Fanuc TP program (LS listing): block_2R_B2_4_Q40_R10.ls

/PROG  block_2R_B2_4_Q40_R10
/ATTR
COMMENT	= "19-04-12 14:24:10";
PROG_SIZE	= 0;
DEFAULT_GROUP	= 1, *, *, *, *;
/APPL
    ARC Welding Equipment: 1, *, *, *, *;
/MN
   1:  CALL HOME_ALL;
   1:  UFRAME_NUM = 1;
   1:  UTOOL_NUM = 3;
   1:  COL GUARD ADJUST 150;
   1:  !Teach Startpoint in PR90;
   1:  !Weld speed R100 in mm/sec;
   1:  !Retraction +Z in R101 in mm;
   1:  !Retraction speed in R102 in %;
   1:  !END_PUB Time in R103;
   1:  !Zeit bis Drahtvorschub R104;
   1:  !Drahtvorschubzeit R105;
   1:  !- Layer/Ebene 1;
   1:  PR[91] = PR[90];
   1:  PR[91,1] = PR[90,1] + 38.877;
   1:  PR[91,2] = PR[90,2] + 1.192;
   1:  PR[91,3] = PR[90,3] + 2.500;
   1:  PR[92] = PR[91];
   1:  PR[92,3] = PR[92,3] + R[101];
   1:J PR[92] R[102]% CNT100;
   1:L PR[91] 100mm/sec FINE RampTo R[100]  Weld Start[1,5.0];
   1:  GO[2]=R[111];
   1:  PR[91,2] = PR[90,2] + 38.792;
   1:L PR[91] R[100]mm/sec CNT100;
   1:  PR[91,1] = PR[90,1] + 1.277;
   1:L PR[91] R[100]mm/sec CNT100;
   1:  PR[91,2] = PR[90,2] + 1.192;
   1:L PR[91] R[100]mm/sec CNT100;
   1:  PR[91,1] = PR[90,1] + 38.877;
   1:L PR[91] R[100]mm/sec CNT100  Weld End[1,5.0,0.2s];
   1:  WAIT R[104];
   1:  PR[92] = PR[91];
   1:  PR[92,3] = PR[92,3] + R[101];
   1:J PR[92] R[102]% CNT100;
   1:  PR[91,1] = PR[90,1] + 36.477;
   1:  PR[91,2] = PR[90,2] + 3.592;
   1:  PR[92] = PR[91];
   1:  PR[92,3] = PR[92,3] + R[101];
   1:J PR[92] R[102]% CNT100;
   1:L PR[91] 100mm/sec FINE RampTo R[100]  Weld Start[1,5.0];
   1:  GO[2]=R[111];
   1:  PR[91,2] = PR[90,2] + 36.392;
   1:L PR[91] R[100]mm/sec CNT100;
   1:  PR[91,1] = PR[90,1] + 3.677;
   1:L PR[91] R[100]mm/sec CNT100;
   1:  PR[91,2] = PR[90,2] + 3.592;
   1:L PR[91] R[100]mm/sec CNT100;
   1:  PR[91,1] = PR[90,1] + 36.477;
   1:L PR[91] R[100]mm/sec CNT100  Weld End[1,5.0,0.2s];
   1:  WAIT R[104];
   1:  PR[92] = PR[91];
   1:  PR[92,3] = PR[92,3] + R[101];
   1:J PR[92] R[102]% CNT100;
   1:  PR[91,1] = PR[90,1] + 25.483;
   1:  PR[91,2] = PR[90,2] + 16.870;
   1:  PR[92] = PR[91];
   1:  PR[92,3] = PR[92,3] + R[101];
   1:J PR[92] R[102]% CNT100;
   1:L PR[91] 100mm/sec FINE RampTo R[100]  Weld Start[1,5.0];
   1:  GO[2]=R[111];
   1:  PR[91,1] = PR[90,1] + 23.198;
   1:  PR[91,2] = PR[90,2] + 14.586;
   1:L PR[91] R[100]mm/sec CNT100;
   1:  PR[91,1] = PR[90,1] + 20.077;
   1:  PR[91,2] = PR[90,2] + 13.750;
   1:L PR[91] R[100]mm/sec CNT100;
   1:  PR[91,1] = PR[90,1] + 16.957;
   1:  PR[91,2] = PR[90,2] + 14.586;
   1:L PR[91] R[100]mm/sec CNT100;
   1:  PR[91,1] = PR[90,1] + 14.672;
   1:  PR[91,2] = PR[90,2] + 16.870;
   1:L PR[91] R[100]mm/sec CNT100;
   1:  PR[91,1] = PR[90,1] + 13.835;
   1:  PR[91,2] = PR[90,2] + 19.992;
   1:L PR[91] R[100]mm/sec CNT100;
   1:  PR[91,1] = PR[90,1] + 14.672;
   1:  PR[91,2] = PR[90,2] + 23.113;
   1:L PR[91] R[100]mm/sec CNT100;
   1:  PR[91,1] = PR[90,1] + 16.957;
   1:  PR[91,2] = PR[90,2] + 25.398;
   1:L PR[91] R[100]mm/sec CNT100;
   1:  PR[91,1] = PR[90,1] + 20.077;
   1:  PR[91,2] = PR[90,2] + 26.234;
   1:L PR[91] R[100]mm/sec CNT100;
   1:  PR[91,1] = PR[90,1] + 23.198;
   1:  PR[91,2] = PR[90,2] + 25.398;
   1:L PR[91] R[100]mm/sec CNT100;
   1:  PR[91,1] = PR[90,1] + 25.483;
   1:  PR[91,2] = PR[90,2] + 23.113;
   1:L PR[91] R[100]mm/sec CNT100;
   1:  PR[91,1] = PR[90,1] + 26.320;
   1:  PR[91,2] = PR[90,2] + 19.992;
   1:L PR[91] R[100]mm/sec CNT100;
   1:  PR[91,1] = PR[90,1] + 25.483;
   1:  PR[91,2] = PR[90,2] + 16.870;
   1:L PR[91] R[100]mm/sec CNT100  Weld End[1,5.0,0.2s];
   1:  WAIT R[104];
   1:  PR[92] = PR[91];
   1:  PR[92,3] = PR[92,3] + R[101];
   1:J PR[92] R[102]% CNT100;
   1:  PR[91,1] = PR[90,1] + 27.635;
   1:  PR[91,2] = PR[90,2] + 15.627;
   1:  PR[92] = PR[91];
   1:  PR[92,3] = PR[92,3] + R[101];
   1:J PR[92] R[102]% CNT100;
   1:L PR[91] 100mm/sec FINE RampTo R[100]  Weld Start[1,5.0];
   1:  GO[2]=R[111];
   1:  PR[91,1] = PR[90,1] + 24.440;
   1:  PR[91,2] = PR[90,2] + 12.434;
   1:L PR[91] R[100]mm/sec CNT100;
   1:  PR[91,1] = PR[90,1] + 20.077;
   1:  PR[91,2] = PR[90,2] + 11.265;
   1:L PR[91] R[100]mm/sec CNT100;
   1:  PR[91,1] = PR[90,1] + 15.715;
   1:  PR[91,2] = PR[90,2] + 12.434;
   1:L PR[91] R[100]mm/sec CNT100;
   1:  PR[91,1] = PR[90,1] + 12.520;
   1:  PR[91,2] = PR[90,2] + 15.627;
   1:L PR[91] R[100]mm/sec CNT100;
   1:  PR[91,1] = PR[90,1] + 11.350;
   1:  PR[91,2] = PR[90,2] + 19.992;
   1:L PR[91] R[100]mm/sec CNT100;
   1:  PR[91,1] = PR[90,1] + 12.520;
   1:  PR[91,2] = PR[90,2] + 24.356;
   1:L PR[91] R[100]mm/sec CNT100;
   1:  PR[91,1] = PR[90,1] + 15.715;
   1:  PR[91,2] = PR[90,2] + 27.550;
   1:L PR[91] R[100]mm/sec CNT100;
   1:  PR[91,1] = PR[90,1] + 20.077;
   1:  PR[91,2] = PR[90,2] + 28.719;
   1:L PR[91] R[100]mm/sec CNT100;
   1:  PR[91,1] = PR[90,1] + 24.440;
   1:  PR[91,2] = PR[90,2] + 27.550;
   1:L PR[91] R[100]mm/sec CNT100;
   1:  PR[91,1] = PR[90,1] + 27.635;
   1:  PR[91,2] = PR[90,2] + 24.356;
   1:L PR[91] R[100]mm/sec CNT100;
   1:  PR[91,1] = PR[90,1] + 28.805;
   1:  PR[91,2] = PR[90,2] + 19.992;
   1:L PR[91] R[100]mm/sec CNT100;
   1:  PR[91,1] = PR[90,1] + 27.635;
   1:  PR[91,2] = PR[90,2] + 15.627;
   1:L PR[91] R[100]mm/sec CNT100  Weld End[1,5.0,0.2s];
   1:  WAIT R[104];
   1:  PR[92] = PR[91];
   1:  PR[92,3] = PR[92,3] + R[101];
   1:J PR[92] R[102]% CNT100;
   1:  PR[91,1] = PR[90,1] + 29.744;
   1:  PR[91,2] = PR[90,2] + 16.082;
   1:  PR[92] = PR[91];
   1:  PR[92,3] = PR[92,3] + R[101];
   1:J PR[92] R[102]% CNT100;
   1:L PR[91] 100mm/sec FINE RampTo R[100]  Weld Start[1,5.0];
   1:  GO[2]=R[111];
   1:  PR[91,1] = PR[90,1] + 34.557;
   1:  PR[91,2] = PR[90,2] + 20.895;
   1:L PR[91] R[100]mm/sec CNT100;
   1:  PR[91,2] = PR[90,2] + 24.289;
   1:L PR[91] R[100]mm/sec CNT100;
   1:  PR[91,1] = PR[90,1] + 30.680;
   1:  PR[91,2] = PR[90,2] + 20.412;
   1:L PR[91] R[100]mm/sec CNT100;
   1:  PR[91,1] = PR[90,1] + 29.962;
   1:  PR[91,2] = PR[90,2] + 23.088;
   1:L PR[91] R[100]mm/sec CNT100;
   1:  PR[91,1] = PR[90,1] + 34.557;
   1:  PR[91,2] = PR[90,2] + 27.683;
   1:L PR[91] R[100]mm/sec CNT100;
   1:  PR[91,2] = PR[90,2] + 31.078;
   1:L PR[91] R[100]mm/sec CNT100;
   1:  PR[91,1] = PR[90,1] + 29.093;
   1:  PR[91,2] = PR[90,2] + 25.613;
   1:L PR[91] R[100]mm/sec CNT100;
   1:  PR[91,1] = PR[90,1] + 27.396;
   1:  PR[91,2] = PR[90,2] + 27.310;
   1:L PR[91] R[100]mm/sec CNT100;
   1:  PR[91,1] = PR[90,1] + 34.557;
   1:  PR[91,2] = PR[90,2] + 34.472;
   1:L PR[91] R[100]mm/sec CNT100;
   1:  PR[91,1] = PR[90,1] + 31.163;
   1:L PR[91] R[100]mm/sec CNT100;
   1:  PR[91,1] = PR[90,1] + 25.698;
   1:  PR[91,2] = PR[90,2] + 29.007;
   1:L PR[91] R[100]mm/sec CNT100;
   1:  PR[91,1] = PR[90,1] + 25.434;
   1:  PR[91,2] = PR[90,2] + 29.271;
   1:L PR[91] R[100]mm/sec CNT100;
   1:  PR[91,1] = PR[90,1] + 23.174;
   1:  PR[91,2] = PR[90,2] + 29.877;
   1:L PR[91] R[100]mm/sec CNT100;
   1:  PR[91,1] = PR[90,1] + 27.769;
   1:  PR[91,2] = PR[90,2] + 34.472;
   1:L PR[91] R[100]mm/sec CNT100;
   1:  PR[91,1] = PR[90,1] + 24.375;
   1:L PR[91] R[100]mm/sec CNT100;
   1:  PR[91,1] = PR[90,1] + 20.497;
   1:  PR[91,2] = PR[90,2] + 30.594;
   1:L PR[91] R[100]mm/sec CNT100  Weld End[1,5.0,0.2s];
   1:  WAIT R[104];
   1:  PR[92] = PR[91];
   1:  PR[92,3] = PR[92,3] + R[101];
   1:J PR[92] R[102]% CNT100;
   1:  PR[91,1] = PR[90,1] + 7.405;
   1:  PR[91,2] = PR[90,2] + 34.472;
   1:  PR[92] = PR[91];
   1:  PR[92,3] = PR[92,3] + R[101];
   1:J PR[92] R[102]% CNT100;
   1:L PR[91] 100mm/sec FINE RampTo R[100]  Weld Start[1,5.0];
   1:  GO[2]=R[111];
   1:  PR[91,1] = PR[90,1] + 5.597;
   1:  PR[91,2] = PR[90,2] + 32.665;
   1:L PR[91] R[100]mm/sec CNT100;
   1:  PR[91,2] = PR[90,2] + 29.270;
   1:L PR[91] R[100]mm/sec CNT100;
   1:  PR[91,1] = PR[90,1] + 10.799;
   1:  PR[91,2] = PR[90,2] + 34.472;
   1:L PR[91] R[100]mm/sec CNT100;
   1:  PR[91,1] = PR[90,1] + 14.193;
   1:L PR[91] R[100]mm/sec CNT100;
   1:  PR[91,1] = PR[90,1] + 5.597;
   1:  PR[91,2] = PR[90,2] + 25.876;
   1:L PR[91] R[100]mm/sec CNT100;
   1:  PR[91,2] = PR[90,2] + 22.482;
   1:L PR[91] R[100]mm/sec CNT100;
   1:  PR[91,1] = PR[90,1] + 17.587;
   1:  PR[91,2] = PR[90,2] + 34.472;
   1:L PR[91] R[100]mm/sec CNT100;
   1:  PR[91,1] = PR[90,1] + 20.981;
   1:L PR[91] R[100]mm/sec CNT100;
   1:  PR[91,1] = PR[90,1] + 16.168;
   1:  PR[91,2] = PR[90,2] + 29.659;
   1:L PR[91] R[100]mm/sec CNT100;
   1:  PR[91,1] = PR[90,1] + 14.721;
   1:  PR[91,2] = PR[90,2] + 29.271;
   1:L PR[91] R[100]mm/sec CNT100;
   1:  PR[91,1] = PR[90,1] + 10.799;
   1:  PR[91,2] = PR[90,2] + 25.350;
   1:L PR[91] R[100]mm/sec CNT100;
   1:  PR[91,1] = PR[90,1] + 10.410;
   1:  PR[91,2] = PR[90,2] + 23.901;
   1:L PR[91] R[100]mm/sec CNT100;
   1:  PR[91,1] = PR[90,1] + 5.597;
   1:  PR[91,2] = PR[90,2] + 19.088;
   1:L PR[91] R[100]mm/sec CNT100;
   1:  PR[91,2] = PR[90,2] + 15.694;
   1:L PR[91] R[100]mm/sec CNT100;
   1:  PR[91,1] = PR[90,1] + 9.475;
   1:  PR[91,2] = PR[90,2] + 19.572;
   1:L PR[91] R[100]mm/sec CNT100;
   1:  PR[91,1] = PR[90,1] + 10.193;
   1:  PR[91,2] = PR[90,2] + 16.895;
   1:L PR[91] R[100]mm/sec CNT100;
   1:  PR[91,1] = PR[90,1] + 5.597;
   1:  PR[91,2] = PR[90,2] + 12.300;
   1:L PR[91] R[100]mm/sec CNT100;
   1:  PR[91,2] = PR[90,2] + 8.906;
   1:L PR[91] R[100]mm/sec CNT100;
   1:  PR[91,1] = PR[90,1] + 11.062;
   1:  PR[91,2] = PR[90,2] + 14.370;
   1:L PR[91] R[100]mm/sec CNT100;
   1:  PR[91,1] = PR[90,1] + 12.759;
   1:  PR[91,2] = PR[90,2] + 12.673;
   1:L PR[91] R[100]mm/sec CNT100;
   1:  PR[91,1] = PR[90,1] + 5.597;
   1:  PR[91,2] = PR[90,2] + 5.512;
   1:L PR[91] R[100]mm/sec CNT100;
   1:  PR[91,1] = PR[90,1] + 8.992;
   1:L PR[91] R[100]mm/sec CNT100;
   1:  PR[91,1] = PR[90,1] + 14.456;
   1:  PR[91,2] = PR[90,2] + 10.977;
   1:L PR[91] R[100]mm/sec CNT100;
   1:  PR[91,1] = PR[90,1] + 14.721;
   1:  PR[91,2] = PR[90,2] + 10.712;
   1:L PR[91] R[100]mm/sec CNT100;
   1:  PR[91,1] = PR[90,1] + 16.981;
   1:  PR[91,2] = PR[90,2] + 10.107;
   1:L PR[91] R[100]mm/sec CNT100;
   1:  PR[91,1] = PR[90,1] + 12.386;
   1:  PR[91,2] = PR[90,2] + 5.512;
   1:L PR[91] R[100]mm/sec CNT100;
   1:  PR[91,1] = PR[90,1] + 15.780;
   1:L PR[91] R[100]mm/sec CNT100;
   1:  PR[91,1] = PR[90,1] + 19.658;
   1:  PR[91,2] = PR[90,2] + 9.390;
   1:L PR[91] R[100]mm/sec CNT100;
   1:  PR[91,1] = PR[90,1] + 20.077;
   1:  PR[91,2] = PR[90,2] + 9.277;
   1:L PR[91] R[100]mm/sec CNT100;
   1:  PR[91,1] = PR[90,1] + 23.987;
   1:  PR[91,2] = PR[90,2] + 10.324;
   1:L PR[91] R[100]mm/sec CNT100;
   1:  PR[91,1] = PR[90,1] + 19.174;
   1:  PR[91,2] = PR[90,2] + 5.512;
   1:L PR[91] R[100]mm/sec CNT100;
   1:  PR[91,1] = PR[90,1] + 22.568;
   1:L PR[91] R[100]mm/sec CNT100;
   1:  PR[91,1] = PR[90,1] + 34.557;
   1:  PR[91,2] = PR[90,2] + 17.501;
   1:L PR[91] R[100]mm/sec CNT100;
   1:  PR[91,2] = PR[90,2] + 14.107;
   1:L PR[91] R[100]mm/sec CNT100;
   1:  PR[91,1] = PR[90,1] + 25.962;
   1:  PR[91,2] = PR[90,2] + 5.512;
   1:L PR[91] R[100]mm/sec CNT100;
   1:  PR[91,1] = PR[90,1] + 29.356;
   1:L PR[91] R[100]mm/sec CNT100;
   1:  PR[91,1] = PR[90,1] + 34.557;
   1:  PR[91,2] = PR[90,2] + 10.713;
   1:L PR[91] R[100]mm/sec CNT100;
   1:  PR[91,2] = PR[90,2] + 7.319;
   1:L PR[91] R[100]mm/sec CNT100;
   1:  PR[91,1] = PR[90,1] + 32.750;
   1:  PR[91,2] = PR[90,2] + 5.512;
   1:L PR[91] R[100]mm/sec CNT100  Weld End[1,5.0,0.2s];
   1:  WAIT R[104];
   1:  PR[92] = PR[91];
   1:  PR[92,3] = PR[92,3] + R[101];
   1:J PR[92] R[102]% CNT100;
   1:  !- Layer/Ebene 2;
   1:  PR[91] = PR[90];
   1:  PR[91,1] = PR[90,1] + 38.877;
   1:  PR[91,2] = PR[90,2] + 38.792;
   1:  PR[91,3] = PR[90,3] + 5.000;
   1:  PR[92] = PR[91];
   1:  PR[92,3] = PR[92,3] + R[101];
   1:J PR[92] R[102]% CNT100;
   1:L PR[91] 100mm/sec FINE RampTo R[100]  Weld Start[1,5.0];
   1:  GO[2]=R[112];
   1:  PR[91,1] = PR[90,1] + 1.277;
   1:L PR[91] R[100]mm/sec CNT100;
   1:  PR[91,2] = PR[90,2] + 1.192;
   1:L PR[91] R[100]mm/sec CNT100;
   1:  PR[91,1] = PR[90,1] + 38.877;
   1:L PR[91] R[100]mm/sec CNT100;
   1:  PR[91,2] = PR[90,2] + 38.792;
   1:L PR[91] R[100]mm/sec CNT100  Weld End[1,5.0,0.2s];
   1:  WAIT R[104];
   1:  PR[92] = PR[91];
   1:  PR[92,3] = PR[92,3] + R[101];
   1:J PR[92] R[102]% CNT100;
   1:  PR[91,1] = PR[90,1] + 36.477;
   1:  PR[91,2] = PR[90,2] + 36.392;
   1:  PR[92] = PR[91];
   1:  PR[92,3] = PR[92,3] + R[101];
   1:J PR[92] R[102]% CNT100;
   1:L PR[91] 100mm/sec FINE RampTo R[100]  Weld Start[1,5.0];
   1:  GO[2]=R[112];
   1:  PR[91,1] = PR[90,1] + 3.677;
   1:L PR[91] R[100]mm/sec CNT100;
   1:  PR[91,2] = PR[90,2] + 3.592;
   1:L PR[91] R[100]mm/sec CNT100;
   1:  PR[91,1] = PR[90,1] + 36.477;
   1:L PR[91] R[100]mm/sec CNT100;
   1:  PR[91,2] = PR[90,2] + 36.392;
   1:L PR[91] R[100]mm/sec CNT100  Weld End[1,5.0,0.2s];
   1:  WAIT R[104];
   1:  PR[92] = PR[91];
   1:  PR[92,3] = PR[92,3] + R[101];
   1:J PR[92] R[102]% CNT100;
   1:  PR[91,1] = PR[90,1] + 25.483;
   1:  PR[91,2] = PR[90,2] + 23.113;
   1:  PR[92] = PR[91];
   1:  PR[92,3] = PR[92,3] + R[101];
   1:J PR[92] R[102]% CNT100;
   1:L PR[91] 100mm/sec FINE RampTo R[100]  Weld Start[1,5.0];
   1:  GO[2]=R[112];
   1:  PR[91,1] = PR[90,1] + 26.320;
   1:  PR[91,2] = PR[90,2] + 19.992;
   1:L PR[91] R[100]mm/sec CNT100;
   1:  PR[91,1] = PR[90,1] + 25.483;
   1:  PR[91,2] = PR[90,2] + 16.870;
   1:L PR[91] R[100]mm/sec CNT100;
   1:  PR[91,1] = PR[90,1] + 23.198;
   1:  PR[91,2] = PR[90,2] + 14.586;
   1:L PR[91] R[100]mm/sec CNT100;
   1:  PR[91,1] = PR[90,1] + 20.077;
   1:  PR[91,2] = PR[90,2] + 13.750;
   1:L PR[91] R[100]mm/sec CNT100;
   1:  PR[91,1] = PR[90,1] + 16.957;
   1:  PR[91,2] = PR[90,2] + 14.586;
   1:L PR[91] R[100]mm/sec CNT100;
   1:  PR[91,1] = PR[90,1] + 14.672;
   1:  PR[91,2] = PR[90,2] + 16.870;
   1:L PR[91] R[100]mm/sec CNT100;
   1:  PR[91,1] = PR[90,1] + 13.835;
   1:  PR[91,2] = PR[90,2] + 19.992;
   1:L PR[91] R[100]mm/sec CNT100;
   1:  PR[91,1] = PR[90,1] + 14.672;
   1:  PR[91,2] = PR[90,2] + 23.113;
   1:L PR[91] R[100]mm/sec CNT100;
   1:  PR[91,1] = PR[90,1] + 16.957;
   1:  PR[91,2] = PR[90,2] + 25.398;
   1:L PR[91] R[100]mm/sec CNT100;
   1:  PR[91,1] = PR[90,1] + 20.077;
   1:  PR[91,2] = PR[90,2] + 26.234;
   1:L PR[91] R[100]mm/sec CNT100;
   1:  PR[91,1] = PR[90,1] + 23.198;
   1:  PR[91,2] = PR[90,2] + 25.398;
   1:L PR[91] R[100]mm/sec CNT100;
   1:  PR[91,1] = PR[90,1] + 25.483;
   1:  PR[91,2] = PR[90,2] + 23.113;
   1:L PR[91] R[100]mm/sec CNT100  Weld End[1,5.0,0.2s];
   1:  WAIT R[104];
   1:  PR[92] = PR[91];
   1:  PR[92,3] = PR[92,3] + R[101];
   1:J PR[92] R[102]% CNT100;
   1:  PR[91,1] = PR[90,1] + 27.635;
   1:  PR[91,2] = PR[90,2] + 24.356;
   1:  PR[92] = PR[91];
   1:  PR[92,3] = PR[92,3] + R[101];
   1:J PR[92] R[102]% CNT100;
   1:L PR[91] 100mm/sec FINE RampTo R[100]  Weld Start[1,5.0];
   1:  GO[2]=R[112];
   1:  PR[91,1] = PR[90,1] + 28.805;
   1:  PR[91,2] = PR[90,2] + 19.992;
   1:L PR[91] R[100]mm/sec CNT100;
   1:  PR[91,1] = PR[90,1] + 27.635;
   1:  PR[91,2] = PR[90,2] + 15.627;
   1:L PR[91] R[100]mm/sec CNT100;
   1:  PR[91,1] = PR[90,1] + 24.440;
   1:  PR[91,2] = PR[90,2] + 12.434;
   1:L PR[91] R[100]mm/sec CNT100;
   1:  PR[91,1] = PR[90,1] + 20.077;
   1:  PR[91,2] = PR[90,2] + 11.265;
   1:L PR[91] R[100]mm/sec CNT100;
   1:  PR[91,1] = PR[90,1] + 15.715;
   1:  PR[91,2] = PR[90,2] + 12.434;
   1:L PR[91] R[100]mm/sec CNT100;
   1:  PR[91,1] = PR[90,1] + 12.520;
   1:  PR[91,2] = PR[90,2] + 15.627;
   1:L PR[91] R[100]mm/sec CNT100;
   1:  PR[91,1] = PR[90,1] + 11.350;
   1:  PR[91,2] = PR[90,2] + 19.992;
   1:L PR[91] R[100]mm/sec CNT100;
   1:  PR[91,1] = PR[90,1] + 12.520;
   1:  PR[91,2] = PR[90,2] + 24.356;
   1:L PR[91] R[100]mm/sec CNT100;
   1:  PR[91,1] = PR[90,1] + 15.715;
   1:  PR[91,2] = PR[90,2] + 27.550;
   1:L PR[91] R[100]mm/sec CNT100;
   1:  PR[91,1] = PR[90,1] + 20.077;
   1:  PR[91,2] = PR[90,2] + 28.719;
   1:L PR[91] R[100]mm/sec CNT100;
   1:  PR[91,1] = PR[90,1] + 24.440;
   1:  PR[91,2] = PR[90,2] + 27.550;
   1:L PR[91] R[100]mm/sec CNT100;
   1:  PR[91,1] = PR[90,1] + 27.635;
   1:  PR[91,2] = PR[90,2] + 24.356;
   1:L PR[91] R[100]mm/sec CNT100  Weld End[1,5.0,0.2s];
   1:  WAIT R[104];
   1:  PR[92] = PR[91];
   1:  PR[92,3] = PR[92,3] + R[101];
   1:J PR[92] R[102]% CNT100;
   1:  PR[91,1] = PR[90,1] + 30.680;
   1:  PR[91,2] = PR[90,2] + 19.572;
   1:  PR[92] = PR[91];
   1:  PR[92,3] = PR[92,3] + R[101];
   1:J PR[92] R[102]% CNT100;
   1:L PR[91] 100mm/sec FINE RampTo R[100]  Weld Start[1,5.0];
   1:  GO[2]=R[112];
   1:  PR[91,1] = PR[90,1] + 34.557;
   1:  PR[91,2] = PR[90,2] + 15.694;
   1:L PR[91] R[100]mm/sec CNT100;
   1:  PR[91,2] = PR[90,2] + 12.300;
   1:L PR[91] R[100]mm/sec CNT100;
   1:  PR[91,1] = PR[90,1] + 29.962;
   1:  PR[91,2] = PR[90,2] + 16.895;
   1:L PR[91] R[100]mm/sec CNT100;
   1:  PR[91,1] = PR[90,1] + 29.356;
   1:  PR[91,2] = PR[90,2] + 14.633;
   1:L PR[91] R[100]mm/sec CNT100;
   1:  PR[91,1] = PR[90,1] + 29.093;
   1:  PR[91,2] = PR[90,2] + 14.370;
   1:L PR[91] R[100]mm/sec CNT100;
   1:  PR[91,1] = PR[90,1] + 34.557;
   1:  PR[91,2] = PR[90,2] + 8.906;
   1:L PR[91] R[100]mm/sec CNT100;
   1:  PR[91,2] = PR[90,2] + 5.512;
   1:L PR[91] R[100]mm/sec CNT100;
   1:  PR[91,1] = PR[90,1] + 27.396;
   1:  PR[91,2] = PR[90,2] + 12.673;
   1:L PR[91] R[100]mm/sec CNT100;
   1:  PR[91,1] = PR[90,1] + 25.698;
   1:  PR[91,2] = PR[90,2] + 10.977;
   1:L PR[91] R[100]mm/sec CNT100;
   1:  PR[91,1] = PR[90,1] + 31.163;
   1:  PR[91,2] = PR[90,2] + 5.512;
   1:L PR[91] R[100]mm/sec CNT100;
   1:  PR[91,1] = PR[90,1] + 27.769;
   1:L PR[91] R[100]mm/sec CNT100;
   1:  PR[91,1] = PR[90,1] + 23.174;
   1:  PR[91,2] = PR[90,2] + 10.107;
   1:L PR[91] R[100]mm/sec CNT100;
   1:  PR[91,1] = PR[90,1] + 20.497;
   1:  PR[91,2] = PR[90,2] + 9.390;
   1:L PR[91] R[100]mm/sec CNT100;
   1:  PR[91,1] = PR[90,1] + 24.375;
   1:  PR[91,2] = PR[90,2] + 5.512;
   1:L PR[91] R[100]mm/sec CNT100;
   1:  PR[91,1] = PR[90,1] + 20.981;
   1:L PR[91] R[100]mm/sec CNT100;
   1:  PR[91,1] = PR[90,1] + 16.168;
   1:  PR[91,2] = PR[90,2] + 10.324;
   1:L PR[91] R[100]mm/sec CNT100  Weld End[1,5.0,0.2s];
   1:  WAIT R[104];
   1:  PR[92] = PR[91];
   1:  PR[92,3] = PR[92,3] + R[101];
   1:J PR[92] R[102]% CNT100;
   1:  PR[91,1] = PR[90,1] + 5.597;
   1:  PR[91,2] = PR[90,2] + 7.319;
   1:  PR[92] = PR[91];
   1:  PR[92,3] = PR[92,3] + R[101];
   1:J PR[92] R[102]% CNT100;
   1:L PR[91] 100mm/sec FINE RampTo R[100]  Weld Start[1,5.0];
   1:  GO[2]=R[112];
   1:  PR[91,1] = PR[90,1] + 7.405;
   1:  PR[91,2] = PR[90,2] + 5.512;
   1:L PR[91] R[100]mm/sec CNT100;
   1:  PR[91,1] = PR[90,1] + 10.799;
   1:L PR[91] R[100]mm/sec CNT100;
   1:  PR[91,1] = PR[90,1] + 5.597;
   1:  PR[91,2] = PR[90,2] + 10.713;
   1:L PR[91] R[100]mm/sec CNT100;
   1:  PR[91,2] = PR[90,2] + 14.107;
   1:L PR[91] R[100]mm/sec CNT100;
   1:  PR[91,1] = PR[90,1] + 14.193;
   1:  PR[91,2] = PR[90,2] + 5.512;
   1:L PR[91] R[100]mm/sec CNT100;
   1:  PR[91,1] = PR[90,1] + 17.587;
   1:L PR[91] R[100]mm/sec CNT100;
   1:  PR[91,1] = PR[90,1] + 5.597;
   1:  PR[91,2] = PR[90,2] + 17.501;
   1:L PR[91] R[100]mm/sec CNT100;
   1:  PR[91,2] = PR[90,2] + 20.895;
   1:L PR[91] R[100]mm/sec CNT100;
   1:  PR[91,1] = PR[90,1] + 10.410;
   1:  PR[91,2] = PR[90,2] + 16.082;
   1:L PR[91] R[100]mm/sec CNT100;
   1:  PR[91,1] = PR[90,1] + 9.363;
   1:  PR[91,2] = PR[90,2] + 19.992;
   1:L PR[91] R[100]mm/sec CNT100;
   1:  PR[91,1] = PR[90,1] + 9.475;
   1:  PR[91,2] = PR[90,2] + 20.412;
   1:L PR[91] R[100]mm/sec CNT100;
   1:  PR[91,1] = PR[90,1] + 5.597;
   1:  PR[91,2] = PR[90,2] + 24.289;
   1:L PR[91] R[100]mm/sec CNT100;
   1:  PR[91,2] = PR[90,2] + 27.684;
   1:L PR[91] R[100]mm/sec CNT100;
   1:  PR[91,1] = PR[90,1] + 10.193;
   1:  PR[91,2] = PR[90,2] + 23.088;
   1:L PR[91] R[100]mm/sec CNT100;
   1:  PR[91,1] = PR[90,1] + 10.799;
   1:  PR[91,2] = PR[90,2] + 25.350;
   1:L PR[91] R[100]mm/sec CNT100;
   1:  PR[91,1] = PR[90,1] + 11.062;
   1:  PR[91,2] = PR[90,2] + 25.613;
   1:L PR[91] R[100]mm/sec CNT100;
   1:  PR[91,1] = PR[90,1] + 5.597;
   1:  PR[91,2] = PR[90,2] + 31.078;
   1:L PR[91] R[100]mm/sec CNT100;
   1:  PR[91,2] = PR[90,2] + 34.472;
   1:L PR[91] R[100]mm/sec CNT100;
   1:  PR[91,1] = PR[90,1] + 12.759;
   1:  PR[91,2] = PR[90,2] + 27.310;
   1:L PR[91] R[100]mm/sec CNT100;
   1:  PR[91,1] = PR[90,1] + 14.456;
   1:  PR[91,2] = PR[90,2] + 29.007;
   1:L PR[91] R[100]mm/sec CNT100;
   1:  PR[91,1] = PR[90,1] + 8.992;
   1:  PR[91,2] = PR[90,2] + 34.472;
   1:L PR[91] R[100]mm/sec CNT100;
   1:  PR[91,1] = PR[90,1] + 12.386;
   1:L PR[91] R[100]mm/sec CNT100;
   1:  PR[91,1] = PR[90,1] + 16.981;
   1:  PR[91,2] = PR[90,2] + 29.877;
   1:L PR[91] R[100]mm/sec CNT100;
   1:  PR[91,1] = PR[90,1] + 19.658;
   1:  PR[91,2] = PR[90,2] + 30.594;
   1:L PR[91] R[100]mm/sec CNT100;
   1:  PR[91,1] = PR[90,1] + 15.780;
   1:  PR[91,2] = PR[90,2] + 34.472;
   1:L PR[91] R[100]mm/sec CNT100;
   1:  PR[91,1] = PR[90,1] + 19.174;
   1:L PR[91] R[100]mm/sec CNT100;
   1:  PR[91,1] = PR[90,1] + 23.987;
   1:  PR[91,2] = PR[90,2] + 29.659;
   1:L PR[91] R[100]mm/sec CNT100;
   1:  PR[91,1] = PR[90,1] + 25.434;
   1:  PR[91,2] = PR[90,2] + 29.271;
   1:L PR[91] R[100]mm/sec CNT100;
   1:  PR[91,1] = PR[90,1] + 29.356;
   1:  PR[91,2] = PR[90,2] + 25.350;
   1:L PR[91] R[100]mm/sec CNT100;
   1:  PR[91,1] = PR[90,1] + 29.744;
   1:  PR[91,2] = PR[90,2] + 23.901;
   1:L PR[91] R[100]mm/sec CNT100;
   1:  PR[91,1] = PR[90,1] + 34.557;
   1:  PR[91,2] = PR[90,2] + 19.088;
   1:L PR[91] R[100]mm/sec CNT100;
   1:  PR[91,2] = PR[90,2] + 22.482;
   1:L PR[91] R[100]mm/sec CNT100;
   1:  PR[91,1] = PR[90,1] + 22.568;
   1:  PR[91,2] = PR[90,2] + 34.472;
   1:L PR[91] R[100]mm/sec CNT100;
   1:  PR[91,1] = PR[90,1] + 25.962;
   1:L PR[91] R[100]mm/sec CNT100;
   1:  PR[91,1] = PR[90,1] + 34.557;
   1:  PR[91,2] = PR[90,2] + 25.876;
   1:L PR[91] R[100]mm/sec CNT100;
   1:  PR[91,2] = PR[90,2] + 29.271;
   1:L PR[91] R[100]mm/sec CNT100;
   1:  PR[91,1] = PR[90,1] + 29.356;
   1:  PR[91,2] = PR[90,2] + 34.472;
   1:L PR[91] R[100]mm/sec CNT100;
   1:  PR[91,1] = PR[90,1] + 32.750;
   1:L PR[91] R[100]mm/sec CNT100;
   1:  PR[91,1] = PR[90,1] + 34.557;
   1:  PR[91,2] = PR[90,2] + 32.665;
   1:L PR[91] R[100]mm/sec CNT100  Weld End[1,5.0,0.2s];
   1:  WAIT R[104];
   1:  PR[92] = PR[91];
   1:  PR[92,3] = PR[92,3] + R[101];
   1:J PR[92] R[102]% CNT100;
   1:  !- Layer/Ebene 3;
   1:  PR[91] = PR[90];
   1:  PR[91,1] = PR[90,1] + 38.877;
   1:  PR[91,2] = PR[90,2] + 38.792;
   1:  PR[91,3] = PR[90,3] + 7.500;
   1:  PR[92] = PR[91];
   1:  PR[92,3] = PR[92,3] + R[101];
   1:J PR[92] R[102]% CNT100;
   1:L PR[91] 100mm/sec FINE RampTo R[100]  Weld Start[1,5.0];
   1:  GO[2]=R[113];
   1:  PR[91,1] = PR[90,1] + 1.277;
   1:L PR[91] R[100]mm/sec CNT100;
   1:  PR[91,2] = PR[90,2] + 1.192;
   1:L PR[91] R[100]mm/sec CNT100;
   1:  PR[91,1] = PR[90,1] + 38.877;
   1:L PR[91] R[100]mm/sec CNT100;
   1:  PR[91,2] = PR[90,2] + 38.792;
   1:L PR[91] R[100]mm/sec CNT100  Weld End[1,5.0,0.2s];
   1:  WAIT R[104];
   1:  PR[92] = PR[91];
   1:  PR[92,3] = PR[92,3] + R[101];
   1:J PR[92] R[102]% CNT100;
   1:  PR[91,1] = PR[90,1] + 36.477;
   1:  PR[91,2] = PR[90,2] + 36.392;
   1:  PR[92] = PR[91];
   1:  PR[92,3] = PR[92,3] + R[101];
   1:J PR[92] R[102]% CNT100;
   1:L PR[91] 100mm/sec FINE RampTo R[100]  Weld Start[1,5.0];
   1:  GO[2]=R[113];
   1:  PR[91,1] = PR[90,1] + 3.677;
   1:L PR[91] R[100]mm/sec CNT100;
   1:  PR[91,2] = PR[90,2] + 3.592;
   1:L PR[91] R[100]mm/sec CNT100;
   1:  PR[91,1] = PR[90,1] + 36.477;
   1:L PR[91] R[100]mm/sec CNT100;
   1:  PR[91,2] = PR[90,2] + 36.392;
   1:L PR[91] R[100]mm/sec CNT100  Weld End[1,5.0,0.2s];
   1:  WAIT R[104];
   1:  PR[92] = PR[91];
   1:  PR[92,3] = PR[92,3] + R[101];
   1:J PR[92] R[102]% CNT100;
   1:  PR[91,1] = PR[90,1] + 25.483;
   1:  PR[91,2] = PR[90,2] + 23.113;
   1:  PR[92] = PR[91];
   1:  PR[92,3] = PR[92,3] + R[101];
   1:J PR[92] R[102]% CNT100;
   1:L PR[91] 100mm/sec FINE RampTo R[100]  Weld Start[1,5.0];
   1:  GO[2]=R[113];
   1:  PR[91,1] = PR[90,1] + 26.320;
   1:  PR[91,2] = PR[90,2] + 19.992;
   1:L PR[91] R[100]mm/sec CNT100;
   1:  PR[91,1] = PR[90,1] + 25.483;
   1:  PR[91,2] = PR[90,2] + 16.870;
   1:L PR[91] R[100]mm/sec CNT100;
   1:  PR[91,1] = PR[90,1] + 23.198;
   1:  PR[91,2] = PR[90,2] + 14.586;
   1:L PR[91] R[100]mm/sec CNT100;
   1:  PR[91,1] = PR[90,1] + 20.077;
   1:  PR[91,2] = PR[90,2] + 13.750;
   1:L PR[91] R[100]mm/sec CNT100;
   1:  PR[91,1] = PR[90,1] + 16.957;
   1:  PR[91,2] = PR[90,2] + 14.586;
   1:L PR[91] R[100]mm/sec CNT100;
   1:  PR[91,1] = PR[90,1] + 14.672;
   1:  PR[91,2] = PR[90,2] + 16.870;
   1:L PR[91] R[100]mm/sec CNT100;
   1:  PR[91,1] = PR[90,1] + 13.835;
   1:  PR[91,2] = PR[90,2] + 19.992;
   1:L PR[91] R[100]mm/sec CNT100;
   1:  PR[91,1] = PR[90,1] + 14.672;
   1:  PR[91,2] = PR[90,2] + 23.113;
   1:L PR[91] R[100]mm/sec CNT100;
   1:  PR[91,1] = PR[90,1] + 16.957;
   1:  PR[91,2] = PR[90,2] + 25.398;
   1:L PR[91] R[100]mm/sec CNT100;
   1:  PR[91,1] = PR[90,1] + 20.077;
   1:  PR[91,2] = PR[90,2] + 26.234;
   1:L PR[91] R[100]mm/sec CNT100;
   1:  PR[91,1] = PR[90,1] + 23.198;
   1:  PR[91,2] = PR[90,2] + 25.398;
   1:L PR[91] R[100]mm/sec CNT100;
   1:  PR[91,1] = PR[90,1] + 25.483;
   1:  PR[91,2] = PR[90,2] + 23.113;
   1:L PR[91] R[100]mm/sec CNT100  Weld End[1,5.0,0.2s];
   1:  WAIT R[104];
   1:  PR[92] = PR[91];
   1:  PR[92,3] = PR[92,3] + R[101];
   1:J PR[92] R[102]% CNT100;
   1:  PR[91,1] = PR[90,1] + 27.635;
   1:  PR[91,2] = PR[90,2] + 24.356;
   1:  PR[92] = PR[91];
   1:  PR[92,3] = PR[92,3] + R[101];
   1:J PR[92] R[102]% CNT100;
   1:L PR[91] 100mm/sec FINE RampTo R[100]  Weld Start[1,5.0];
   1:  GO[2]=R[113];
   1:  PR[91,1] = PR[90,1] + 28.805;
   1:  PR[91,2] = PR[90,2] + 19.992;
   1:L PR[91] R[100]mm/sec CNT100;
   1:  PR[91,1] = PR[90,1] + 27.635;
   1:  PR[91,2] = PR[90,2] + 15.627;
   1:L PR[91] R[100]mm/sec CNT100;
   1:  PR[91,1] = PR[90,1] + 24.440;
   1:  PR[91,2] = PR[90,2] + 12.434;
   1:L PR[91] R[100]mm/sec CNT100;
   1:  PR[91,1] = PR[90,1] + 20.077;
   1:  PR[91,2] = PR[90,2] + 11.265;
   1:L PR[91] R[100]mm/sec CNT100;
   1:  PR[91,1] = PR[90,1] + 15.715;
   1:  PR[91,2] = PR[90,2] + 12.434;
   1:L PR[91] R[100]mm/sec CNT100;
   1:  PR[91,1] = PR[90,1] + 12.520;
   1:  PR[91,2] = PR[90,2] + 15.627;
   1:L PR[91] R[100]mm/sec CNT100;
   1:  PR[91,1] = PR[90,1] + 11.350;
   1:  PR[91,2] = PR[90,2] + 19.992;
   1:L PR[91] R[100]mm/sec CNT100;
   1:  PR[91,1] = PR[90,1] + 12.520;
   1:  PR[91,2] = PR[90,2] + 24.356;
   1:L PR[91] R[100]mm/sec CNT100;
   1:  PR[91,1] = PR[90,1] + 15.715;
   1:  PR[91,2] = PR[90,2] + 27.550;
   1:L PR[91] R[100]mm/sec CNT100;
   1:  PR[91,1] = PR[90,1] + 20.077;
   1:  PR[91,2] = PR[90,2] + 28.719;
   1:L PR[91] R[100]mm/sec CNT100;
   1:  PR[91,1] = PR[90,1] + 24.440;
   1:  PR[91,2] = PR[90,2] + 27.550;
   1:L PR[91] R[100]mm/sec CNT100;
   1:  PR[91,1] = PR[90,1] + 27.635;
   1:  PR[91,2] = PR[90,2] + 24.356;
   1:L PR[91] R[100]mm/sec CNT100  Weld End[1,5.0,0.2s];
   1:  WAIT R[104];
   1:  PR[92] = PR[91];
   1:  PR[92,3] = PR[92,3] + R[101];
   1:J PR[92] R[102]% CNT100;
   1:  PR[91,1] = PR[90,1] + 29.744;
   1:  PR[91,2] = PR[90,2] + 16.082;
   1:  PR[92] = PR[91];
   1:  PR[92,3] = PR[92,3] + R[101];
   1:J PR[92] R[102]% CNT100;
   1:L PR[91] 100mm/sec FINE RampTo R[100]  Weld Start[1,5.0];
   1:  GO[2]=R[113];
   1:  PR[91,1] = PR[90,1] + 34.557;
   1:  PR[91,2] = PR[90,2] + 20.895;
   1:L PR[91] R[100]mm/sec CNT100;
   1:  PR[91,2] = PR[90,2] + 24.289;
   1:L PR[91] R[100]mm/sec CNT100;
   1:  PR[91,1] = PR[90,1] + 30.680;
   1:  PR[91,2] = PR[90,2] + 20.412;
   1:L PR[91] R[100]mm/sec CNT100;
   1:  PR[91,1] = PR[90,1] + 29.962;
   1:  PR[91,2] = PR[90,2] + 23.088;
   1:L PR[91] R[100]mm/sec CNT100;
   1:  PR[91,1] = PR[90,1] + 34.557;
   1:  PR[91,2] = PR[90,2] + 27.683;
   1:L PR[91] R[100]mm/sec CNT100;
   1:  PR[91,2] = PR[90,2] + 31.078;
   1:L PR[91] R[100]mm/sec CNT100;
   1:  PR[91,1] = PR[90,1] + 29.093;
   1:  PR[91,2] = PR[90,2] + 25.613;
   1:L PR[91] R[100]mm/sec CNT100;
   1:  PR[91,1] = PR[90,1] + 27.396;
   1:  PR[91,2] = PR[90,2] + 27.310;
   1:L PR[91] R[100]mm/sec CNT100;
   1:  PR[91,1] = PR[90,1] + 34.557;
   1:  PR[91,2] = PR[90,2] + 34.472;
   1:L PR[91] R[100]mm/sec CNT100;
   1:  PR[91,1] = PR[90,1] + 31.163;
   1:L PR[91] R[100]mm/sec CNT100;
   1:  PR[91,1] = PR[90,1] + 25.698;
   1:  PR[91,2] = PR[90,2] + 29.007;
   1:L PR[91] R[100]mm/sec CNT100;
   1:  PR[91,1] = PR[90,1] + 25.434;
   1:  PR[91,2] = PR[90,2] + 29.271;
   1:L PR[91] R[100]mm/sec CNT100;
   1:  PR[91,1] = PR[90,1] + 23.174;
   1:  PR[91,2] = PR[90,2] + 29.877;
   1:L PR[91] R[100]mm/sec CNT100;
   1:  PR[91,1] = PR[90,1] + 27.769;
   1:  PR[91,2] = PR[90,2] + 34.472;
   1:L PR[91] R[100]mm/sec CNT100;
   1:  PR[91,1] = PR[90,1] + 24.375;
   1:L PR[91] R[100]mm/sec CNT100;
   1:  PR[91,1] = PR[90,1] + 20.497;
   1:  PR[91,2] = PR[90,2] + 30.594;
   1:L PR[91] R[100]mm/sec CNT100  Weld End[1,5.0,0.2s];
   1:  WAIT R[104];
   1:  PR[92] = PR[91];
   1:  PR[92,3] = PR[92,3] + R[101];
   1:J PR[92] R[102]% CNT100;
   1:  PR[91,1] = PR[90,1] + 7.405;
   1:  PR[91,2] = PR[90,2] + 34.472;
   1:  PR[92] = PR[91];
   1:  PR[92,3] = PR[92,3] + R[101];
   1:J PR[92] R[102]% CNT100;
   1:L PR[91] 100mm/sec FINE RampTo R[100]  Weld Start[1,5.0];
   1:  GO[2]=R[113];
   1:  PR[91,1] = PR[90,1] + 5.597;
   1:  PR[91,2] = PR[90,2] + 32.665;
   1:L PR[91] R[100]mm/sec CNT100;
   1:  PR[91,2] = PR[90,2] + 29.270;
   1:L PR[91] R[100]mm/sec CNT100;
   1:  PR[91,1] = PR[90,1] + 10.799;
   1:  PR[91,2] = PR[90,2] + 34.472;
   1:L PR[91] R[100]mm/sec CNT100;
   1:  PR[91,1] = PR[90,1] + 14.193;
   1:L PR[91] R[100]mm/sec CNT100;
   1:  PR[91,1] = PR[90,1] + 5.597;
   1:  PR[91,2] = PR[90,2] + 25.876;
   1:L PR[91] R[100]mm/sec CNT100;
   1:  PR[91,2] = PR[90,2] + 22.482;
   1:L PR[91] R[100]mm/sec CNT100;
   1:  PR[91,1] = PR[90,1] + 17.587;
   1:  PR[91,2] = PR[90,2] + 34.472;
   1:L PR[91] R[100]mm/sec CNT100;
   1:  PR[91,1] = PR[90,1] + 20.981;
   1:L PR[91] R[100]mm/sec CNT100;
   1:  PR[91,1] = PR[90,1] + 16.168;
   1:  PR[91,2] = PR[90,2] + 29.659;
   1:L PR[91] R[100]mm/sec CNT100;
   1:  PR[91,1] = PR[90,1] + 14.721;
   1:  PR[91,2] = PR[90,2] + 29.271;
   1:L PR[91] R[100]mm/sec CNT100;
   1:  PR[91,1] = PR[90,1] + 10.799;
   1:  PR[91,2] = PR[90,2] + 25.350;
   1:L PR[91] R[100]mm/sec CNT100;
   1:  PR[91,1] = PR[90,1] + 10.410;
   1:  PR[91,2] = PR[90,2] + 23.901;
   1:L PR[91] R[100]mm/sec CNT100;
   1:  PR[91,1] = PR[90,1] + 5.597;
   1:  PR[91,2] = PR[90,2] + 19.088;
   1:L PR[91] R[100]mm/sec CNT100;
   1:  PR[91,2] = PR[90,2] + 15.694;
   1:L PR[91] R[100]mm/sec CNT100;
   1:  PR[91,1] = PR[90,1] + 9.475;
   1:  PR[91,2] = PR[90,2] + 19.572;
   1:L PR[91] R[100]mm/sec CNT100;
   1:  PR[91,1] = PR[90,1] + 10.193;
   1:  PR[91,2] = PR[90,2] + 16.895;
   1:L PR[91] R[100]mm/sec CNT100;
   1:  PR[91,1] = PR[90,1] + 5.597;
   1:  PR[91,2] = PR[90,2] + 12.300;
   1:L PR[91] R[100]mm/sec CNT100;
   1:  PR[91,2] = PR[90,2] + 8.906;
   1:L PR[91] R[100]mm/sec CNT100;
   1:  PR[91,1] = PR[90,1] + 11.062;
   1:  PR[91,2] = PR[90,2] + 14.370;
   1:L PR[91] R[100]mm/sec CNT100;
   1:  PR[91,1] = PR[90,1] + 12.759;
   1:  PR[91,2] = PR[90,2] + 12.673;
   1:L PR[91] R[100]mm/sec CNT100;
   1:  PR[91,1] = PR[90,1] + 5.597;
   1:  PR[91,2] = PR[90,2] + 5.512;
   1:L PR[91] R[100]mm/sec CNT100;
   1:  PR[91,1] = PR[90,1] + 8.992;
   1:L PR[91] R[100]mm/sec CNT100;
   1:  PR[91,1] = PR[90,1] + 14.456;
   1:  PR[91,2] = PR[90,2] + 10.977;
   1:L PR[91] R[100]mm/sec CNT100;
   1:  PR[91,1] = PR[90,1] + 14.721;
   1:  PR[91,2] = PR[90,2] + 10.712;
   1:L PR[91] R[100]mm/sec CNT100;
   1:  PR[91,1] = PR[90,1] + 16.981;
   1:  PR[91,2] = PR[90,2] + 10.107;
   1:L PR[91] R[100]mm/sec CNT100;
   1:  PR[91,1] = PR[90,1] + 12.386;
   1:  PR[91,2] = PR[90,2] + 5.512;
   1:L PR[91] R[100]mm/sec CNT100;
   1:  PR[91,1] = PR[90,1] + 15.780;
   1:L PR[91] R[100]mm/sec CNT100;
   1:  PR[91,1] = PR[90,1] + 19.658;
   1:  PR[91,2] = PR[90,2] + 9.390;
   1:L PR[91] R[100]mm/sec CNT100;
   1:  PR[91,1] = PR[90,1] + 20.077;
   1:  PR[91,2] = PR[90,2] + 9.277;
   1:L PR[91] R[100]mm/sec CNT100;
   1:  PR[91,1] = PR[90,1] + 23.987;
   1:  PR[91,2] = PR[90,2] + 10.324;
   1:L PR[91] R[100]mm/sec CNT100;
   1:  PR[91,1] = PR[90,1] + 19.174;
   1:  PR[91,2] = PR[90,2] + 5.512;
   1:L PR[91] R[100]mm/sec CNT100;
   1:  PR[91,1] = PR[90,1] + 22.568;
   1:L PR[91] R[100]mm/sec CNT100;
   1:  PR[91,1] = PR[90,1] + 34.557;
   1:  PR[91,2] = PR[90,2] + 17.501;
   1:L PR[91] R[100]mm/sec CNT100;
   1:  PR[91,2] = PR[90,2] + 14.107;
   1:L PR[91] R[100]mm/sec CNT100;
   1:  PR[91,1] = PR[90,1] + 25.962;
   1:  PR[91,2] = PR[90,2] + 5.512;
   1:L PR[91] R[100]mm/sec CNT100;
   1:  PR[91,1] = PR[90,1] + 29.356;
   1:L PR[91] R[100]mm/sec CNT100;
   1:  PR[91,1] = PR[90,1] + 34.557;
   1:  PR[91,2] = PR[90,2] + 10.713;
   1:L PR[91] R[100]mm/sec CNT100;
   1:  PR[91,2] = PR[90,2] + 7.319;
   1:L PR[91] R[100]mm/sec CNT100;
   1:  PR[91,1] = PR[90,1] + 32.750;
   1:  PR[91,2] = PR[90,2] + 5.512;
   1:L PR[91] R[100]mm/sec CNT100  Weld End[1,5.0,0.2s];
   1:  WAIT R[104];
   1:  PR[92] = PR[91];
   1:  PR[92,3] = PR[92,3] + R[101];
   1:J PR[92] R[102]% CNT100;
   1:  !- Layer/Ebene 4;
   1:  PR[91] = PR[90];
   1:  PR[91,1] = PR[90,1] + 1.277;
   1:  PR[91,2] = PR[90,2] + 1.192;
   1:  PR[91,3] = PR[90,3] + 10.000;
   1:  PR[92] = PR[91];
   1:  PR[92,3] = PR[92,3] + R[101];
   1:J PR[92] R[102]% CNT100;
   1:L PR[91] 100mm/sec FINE RampTo R[100]  Weld Start[1,5.0];
   1:  GO[2]=R[113];
   1:  PR[91,1] = PR[90,1] + 38.877;
   1:L PR[91] R[100]mm/sec CNT100;
   1:  PR[91,2] = PR[90,2] + 38.792;
   1:L PR[91] R[100]mm/sec CNT100;
   1:  PR[91,1] = PR[90,1] + 1.277;
   1:L PR[91] R[100]mm/sec CNT100;
   1:  PR[91,2] = PR[90,2] + 1.192;
   1:L PR[91] R[100]mm/sec CNT100  Weld End[1,5.0,0.2s];
   1:  WAIT R[104];
   1:  PR[92] = PR[91];
   1:  PR[92,3] = PR[92,3] + R[101];
   1:J PR[92] R[102]% CNT100;
   1:  PR[91,1] = PR[90,1] + 3.677;
   1:  PR[91,2] = PR[90,2] + 3.592;
   1:  PR[92] = PR[91];
   1:  PR[92,3] = PR[92,3] + R[101];
   1:J PR[92] R[102]% CNT100;
   1:L PR[91] 100mm/sec FINE RampTo R[100]  Weld Start[1,5.0];
   1:  GO[2]=R[113];
   1:  PR[91,1] = PR[90,1] + 36.477;
   1:L PR[91] R[100]mm/sec CNT100;
   1:  PR[91,2] = PR[90,2] + 36.392;
   1:L PR[91] R[100]mm/sec CNT100;
   1:  PR[91,1] = PR[90,1] + 3.677;
   1:L PR[91] R[100]mm/sec CNT100;
   1:  PR[91,2] = PR[90,2] + 3.592;
   1:L PR[91] R[100]mm/sec CNT100  Weld End[1,5.0,0.2s];
   1:  WAIT R[104];
   1:  PR[92] = PR[91];
   1:  PR[92,3] = PR[92,3] + R[101];
   1:J PR[92] R[102]% CNT100;
   1:  PR[91,1] = PR[90,1] + 14.672;
   1:  PR[91,2] = PR[90,2] + 16.870;
   1:  PR[92] = PR[91];
   1:  PR[92,3] = PR[92,3] + R[101];
   1:J PR[92] R[102]% CNT100;
   1:L PR[91] 100mm/sec FINE RampTo R[100]  Weld Start[1,5.0];
   1:  GO[2]=R[113];
   1:  PR[91,1] = PR[90,1] + 13.835;
   1:  PR[91,2] = PR[90,2] + 19.992;
   1:L PR[91] R[100]mm/sec CNT100;
   1:  PR[91,1] = PR[90,1] + 14.672;
   1:  PR[91,2] = PR[90,2] + 23.113;
   1:L PR[91] R[100]mm/sec CNT100;
   1:  PR[91,1] = PR[90,1] + 16.957;
   1:  PR[91,2] = PR[90,2] + 25.398;
   1:L PR[91] R[100]mm/sec CNT100;
   1:  PR[91,1] = PR[90,1] + 20.077;
   1:  PR[91,2] = PR[90,2] + 26.234;
   1:L PR[91] R[100]mm/sec CNT100;
   1:  PR[91,1] = PR[90,1] + 23.198;
   1:  PR[91,2] = PR[90,2] + 25.398;
   1:L PR[91] R[100]mm/sec CNT100;
   1:  PR[91,1] = PR[90,1] + 25.483;
   1:  PR[91,2] = PR[90,2] + 23.113;
   1:L PR[91] R[100]mm/sec CNT100;
   1:  PR[91,1] = PR[90,1] + 26.320;
   1:  PR[91,2] = PR[90,2] + 19.992;
   1:L PR[91] R[100]mm/sec CNT100;
   1:  PR[91,1] = PR[90,1] + 25.483;
   1:  PR[91,2] = PR[90,2] + 16.870;
   1:L PR[91] R[100]mm/sec CNT100;
   1:  PR[91,1] = PR[90,1] + 23.198;
   1:  PR[91,2] = PR[90,2] + 14.586;
   1:L PR[91] R[100]mm/sec CNT100;
   1:  PR[91,1] = PR[90,1] + 20.077;
   1:  PR[91,2] = PR[90,2] + 13.750;
   1:L PR[91] R[100]mm/sec CNT100;
   1:  PR[91,1] = PR[90,1] + 16.957;
   1:  PR[91,2] = PR[90,2] + 14.586;
   1:L PR[91] R[100]mm/sec CNT100;
   1:  PR[91,1] = PR[90,1] + 14.672;
   1:  PR[91,2] = PR[90,2] + 16.870;
   1:L PR[91] R[100]mm/sec CNT100  Weld End[1,5.0,0.2s];
   1:  WAIT R[104];
   1:  PR[92] = PR[91];
   1:  PR[92,3] = PR[92,3] + R[101];
   1:J PR[92] R[102]% CNT100;
   1:  PR[91,1] = PR[90,1] + 12.520;
   1:  PR[91,2] = PR[90,2] + 15.627;
   1:  PR[92] = PR[91];
   1:  PR[92,3] = PR[92,3] + R[101];
   1:J PR[92] R[102]% CNT100;
   1:L PR[91] 100mm/sec FINE RampTo R[100]  Weld Start[1,5.0];
   1:  GO[2]=R[113];
   1:  PR[91,1] = PR[90,1] + 11.350;
   1:  PR[91,2] = PR[90,2] + 19.992;
   1:L PR[91] R[100]mm/sec CNT100;
   1:  PR[91,1] = PR[90,1] + 12.520;
   1:  PR[91,2] = PR[90,2] + 24.356;
   1:L PR[91] R[100]mm/sec CNT100;
   1:  PR[91,1] = PR[90,1] + 15.715;
   1:  PR[91,2] = PR[90,2] + 27.550;
   1:L PR[91] R[100]mm/sec CNT100;
   1:  PR[91,1] = PR[90,1] + 20.077;
   1:  PR[91,2] = PR[90,2] + 28.719;
   1:L PR[91] R[100]mm/sec CNT100;
   1:  PR[91,1] = PR[90,1] + 24.440;
   1:  PR[91,2] = PR[90,2] + 27.550;
   1:L PR[91] R[100]mm/sec CNT100;
   1:  PR[91,1] = PR[90,1] + 27.635;
   1:  PR[91,2] = PR[90,2] + 24.356;
   1:L PR[91] R[100]mm/sec CNT100;
   1:  PR[91,1] = PR[90,1] + 28.805;
   1:  PR[91,2] = PR[90,2] + 19.992;
   1:L PR[91] R[100]mm/sec CNT100;
   1:  PR[91,1] = PR[90,1] + 27.635;
   1:  PR[91,2] = PR[90,2] + 15.627;
   1:L PR[91] R[100]mm/sec CNT100;
   1:  PR[91,1] = PR[90,1] + 24.440;
   1:  PR[91,2] = PR[90,2] + 12.434;
   1:L PR[91] R[100]mm/sec CNT100;
   1:  PR[91,1] = PR[90,1] + 20.077;
   1:  PR[91,2] = PR[90,2] + 11.265;
   1:L PR[91] R[100]mm/sec CNT100;
   1:  PR[91,1] = PR[90,1] + 15.715;
   1:  PR[91,2] = PR[90,2] + 12.434;
   1:L PR[91] R[100]mm/sec CNT100;
   1:  PR[91,1] = PR[90,1] + 12.520;
   1:  PR[91,2] = PR[90,2] + 15.627;
   1:L PR[91] R[100]mm/sec CNT100  Weld End[1,5.0,0.2s];
   1:  WAIT R[104];
   1:  PR[92] = PR[91];
   1:  PR[92,3] = PR[92,3] + R[101];
   1:J PR[92] R[102]% CNT100;
   1:  PR[91,1] = PR[90,1] + 16.168;
   1:  PR[91,2] = PR[90,2] + 10.324;
   1:  PR[92] = PR[91];
   1:  PR[92,3] = PR[92,3] + R[101];
   1:J PR[92] R[102]% CNT100;
   1:L PR[91] 100mm/sec FINE RampTo R[100]  Weld Start[1,5.0];
   1:  GO[2]=R[113];
   1:  PR[91,1] = PR[90,1] + 20.981;
   1:  PR[91,2] = PR[90,2] + 5.512;
   1:L PR[91] R[100]mm/sec CNT100;
   1:  PR[91,1] = PR[90,1] + 24.375;
   1:L PR[91] R[100]mm/sec CNT100;
   1:  PR[91,1] = PR[90,1] + 20.497;
   1:  PR[91,2] = PR[90,2] + 9.390;
   1:L PR[91] R[100]mm/sec CNT100;
   1:  PR[91,1] = PR[90,1] + 23.174;
   1:  PR[91,2] = PR[90,2] + 10.107;
   1:L PR[91] R[100]mm/sec CNT100;
   1:  PR[91,1] = PR[90,1] + 27.769;
   1:  PR[91,2] = PR[90,2] + 5.512;
   1:L PR[91] R[100]mm/sec CNT100;
   1:  PR[91,1] = PR[90,1] + 31.163;
   1:L PR[91] R[100]mm/sec CNT100;
   1:  PR[91,1] = PR[90,1] + 25.698;
   1:  PR[91,2] = PR[90,2] + 10.977;
   1:L PR[91] R[100]mm/sec CNT100;
   1:  PR[91,1] = PR[90,1] + 27.396;
   1:  PR[91,2] = PR[90,2] + 12.673;
   1:L PR[91] R[100]mm/sec CNT100;
   1:  PR[91,1] = PR[90,1] + 34.557;
   1:  PR[91,2] = PR[90,2] + 5.512;
   1:L PR[91] R[100]mm/sec CNT100;
   1:  PR[91,2] = PR[90,2] + 8.906;
   1:L PR[91] R[100]mm/sec CNT100;
   1:  PR[91,1] = PR[90,1] + 29.093;
   1:  PR[91,2] = PR[90,2] + 14.370;
   1:L PR[91] R[100]mm/sec CNT100;
   1:  PR[91,1] = PR[90,1] + 29.356;
   1:  PR[91,2] = PR[90,2] + 14.633;
   1:L PR[91] R[100]mm/sec CNT100;
   1:  PR[91,1] = PR[90,1] + 29.962;
   1:  PR[91,2] = PR[90,2] + 16.895;
   1:L PR[91] R[100]mm/sec CNT100;
   1:  PR[91,1] = PR[90,1] + 34.557;
   1:  PR[91,2] = PR[90,2] + 12.300;
   1:L PR[91] R[100]mm/sec CNT100;
   1:  PR[91,2] = PR[90,2] + 15.694;
   1:L PR[91] R[100]mm/sec CNT100;
   1:  PR[91,1] = PR[90,1] + 30.680;
   1:  PR[91,2] = PR[90,2] + 19.572;
   1:L PR[91] R[100]mm/sec CNT100  Weld End[1,5.0,0.2s];
   1:  WAIT R[104];
   1:  PR[92] = PR[91];
   1:  PR[92,3] = PR[92,3] + R[101];
   1:J PR[92] R[102]% CNT100;
   1:  PR[91,1] = PR[90,1] + 34.557;
   1:  PR[91,2] = PR[90,2] + 32.665;
   1:  PR[92] = PR[91];
   1:  PR[92,3] = PR[92,3] + R[101];
   1:J PR[92] R[102]% CNT100;
   1:L PR[91] 100mm/sec FINE RampTo R[100]  Weld Start[1,5.0];
   1:  GO[2]=R[113];
   1:  PR[91,1] = PR[90,1] + 32.750;
   1:  PR[91,2] = PR[90,2] + 34.472;
   1:L PR[91] R[100]mm/sec CNT100;
   1:  PR[91,1] = PR[90,1] + 29.356;
   1:L PR[91] R[100]mm/sec CNT100;
   1:  PR[91,1] = PR[90,1] + 34.557;
   1:  PR[91,2] = PR[90,2] + 29.271;
   1:L PR[91] R[100]mm/sec CNT100;
   1:  PR[91,2] = PR[90,2] + 25.876;
   1:L PR[91] R[100]mm/sec CNT100;
   1:  PR[91,1] = PR[90,1] + 25.962;
   1:  PR[91,2] = PR[90,2] + 34.472;
   1:L PR[91] R[100]mm/sec CNT100;
   1:  PR[91,1] = PR[90,1] + 22.568;
   1:L PR[91] R[100]mm/sec CNT100;
   1:  PR[91,1] = PR[90,1] + 34.557;
   1:  PR[91,2] = PR[90,2] + 22.482;
   1:L PR[91] R[100]mm/sec CNT100;
   1:  PR[91,2] = PR[90,2] + 19.088;
   1:L PR[91] R[100]mm/sec CNT100;
   1:  PR[91,1] = PR[90,1] + 29.744;
   1:  PR[91,2] = PR[90,2] + 23.901;
   1:L PR[91] R[100]mm/sec CNT100;
   1:  PR[91,1] = PR[90,1] + 29.356;
   1:  PR[91,2] = PR[90,2] + 25.350;
   1:L PR[91] R[100]mm/sec CNT100;
   1:  PR[91,1] = PR[90,1] + 25.434;
   1:  PR[91,2] = PR[90,2] + 29.271;
   1:L PR[91] R[100]mm/sec CNT100;
   1:  PR[91,1] = PR[90,1] + 23.987;
   1:  PR[91,2] = PR[90,2] + 29.659;
   1:L PR[91] R[100]mm/sec CNT100;
   1:  PR[91,1] = PR[90,1] + 19.174;
   1:  PR[91,2] = PR[90,2] + 34.472;
   1:L PR[91] R[100]mm/sec CNT100;
   1:  PR[91,1] = PR[90,1] + 15.780;
   1:L PR[91] R[100]mm/sec CNT100;
   1:  PR[91,1] = PR[90,1] + 19.658;
   1:  PR[91,2] = PR[90,2] + 30.594;
   1:L PR[91] R[100]mm/sec CNT100;
   1:  PR[91,1] = PR[90,1] + 16.981;
   1:  PR[91,2] = PR[90,2] + 29.877;
   1:L PR[91] R[100]mm/sec CNT100;
   1:  PR[91,1] = PR[90,1] + 12.386;
   1:  PR[91,2] = PR[90,2] + 34.472;
   1:L PR[91] R[100]mm/sec CNT100;
   1:  PR[91,1] = PR[90,1] + 8.992;
   1:L PR[91] R[100]mm/sec CNT100;
   1:  PR[91,1] = PR[90,1] + 14.456;
   1:  PR[91,2] = PR[90,2] + 29.007;
   1:L PR[91] R[100]mm/sec CNT100;
   1:  PR[91,1] = PR[90,1] + 12.759;
   1:  PR[91,2] = PR[90,2] + 27.310;
   1:L PR[91] R[100]mm/sec CNT100;
   1:  PR[91,1] = PR[90,1] + 5.597;
   1:  PR[91,2] = PR[90,2] + 34.472;
   1:L PR[91] R[100]mm/sec CNT100;
   1:  PR[91,2] = PR[90,2] + 31.078;
   1:L PR[91] R[100]mm/sec CNT100;
   1:  PR[91,1] = PR[90,1] + 11.062;
   1:  PR[91,2] = PR[90,2] + 25.613;
   1:L PR[91] R[100]mm/sec CNT100;
   1:  PR[91,1] = PR[90,1] + 10.799;
   1:  PR[91,2] = PR[90,2] + 25.350;
   1:L PR[91] R[100]mm/sec CNT100;
   1:  PR[91,1] = PR[90,1] + 10.193;
   1:  PR[91,2] = PR[90,2] + 23.088;
   1:L PR[91] R[100]mm/sec CNT100;
   1:  PR[91,1] = PR[90,1] + 5.597;
   1:  PR[91,2] = PR[90,2] + 27.684;
   1:L PR[91] R[100]mm/sec CNT100;
   1:  PR[91,2] = PR[90,2] + 24.289;
   1:L PR[91] R[100]mm/sec CNT100;
   1:  PR[91,1] = PR[90,1] + 9.475;
   1:  PR[91,2] = PR[90,2] + 20.412;
   1:L PR[91] R[100]mm/sec CNT100;
   1:  PR[91,1] = PR[90,1] + 9.363;
   1:  PR[91,2] = PR[90,2] + 19.992;
   1:L PR[91] R[100]mm/sec CNT100;
   1:  PR[91,1] = PR[90,1] + 10.410;
   1:  PR[91,2] = PR[90,2] + 16.082;
   1:L PR[91] R[100]mm/sec CNT100;
   1:  PR[91,1] = PR[90,1] + 5.597;
   1:  PR[91,2] = PR[90,2] + 20.895;
   1:L PR[91] R[100]mm/sec CNT100;
   1:  PR[91,2] = PR[90,2] + 17.501;
   1:L PR[91] R[100]mm/sec CNT100;
   1:  PR[91,1] = PR[90,1] + 17.587;
   1:  PR[91,2] = PR[90,2] + 5.512;
   1:L PR[91] R[100]mm/sec CNT100;
   1:  PR[91,1] = PR[90,1] + 14.193;
   1:L PR[91] R[100]mm/sec CNT100;
   1:  PR[91,1] = PR[90,1] + 5.597;
   1:  PR[91,2] = PR[90,2] + 14.107;
   1:L PR[91] R[100]mm/sec CNT100;
   1:  PR[91,2] = PR[90,2] + 10.713;
   1:L PR[91] R[100]mm/sec CNT100;
   1:  PR[91,1] = PR[90,1] + 10.799;
   1:  PR[91,2] = PR[90,2] + 5.512;
   1:L PR[91] R[100]mm/sec CNT100;
   1:  PR[91,1] = PR[90,1] + 7.405;
   1:L PR[91] R[100]mm/sec CNT100;
   1:  PR[91,1] = PR[90,1] + 5.597;
   1:  PR[91,2] = PR[90,2] + 7.319;
   1:L PR[91] R[100]mm/sec CNT100  Weld End[1,5.0,0.2s];
   1:  WAIT R[104];
   1:  PR[92] = PR[91];
   1:  PR[92,3] = PR[92,3] + R[101];
   1:J PR[92] R[102]% CNT100;
   1:  !- Layer/Ebene 5;
   1:  PR[91] = PR[90];
   1:  PR[91,1] = PR[90,1] + 38.877;
   1:  PR[91,2] = PR[90,2] + 38.792;
   1:  PR[91,3] = PR[90,3] + 12.500;
   1:  PR[92] = PR[91];
   1:  PR[92,3] = PR[92,3] + R[101];
   1:J PR[92] R[102]% CNT100;
   1:L PR[91] 100mm/sec FINE RampTo R[100]  Weld Start[1,5.0];
   1:  GO[2]=R[113];
   1:  PR[91,1] = PR[90,1] + 1.277;
   1:L PR[91] R[100]mm/sec CNT100;
   1:  PR[91,2] = PR[90,2] + 1.192;
   1:L PR[91] R[100]mm/sec CNT100;
   1:  PR[91,1] = PR[90,1] + 38.877;
   1:L PR[91] R[100]mm/sec CNT100;
   1:  PR[91,2] = PR[90,2] + 38.792;
   1:L PR[91] R[100]mm/sec CNT100  Weld End[1,5.0,0.2s];
   1:  WAIT R[104];
   1:  PR[92] = PR[91];
   1:  PR[92,3] = PR[92,3] + R[101];
   1:J PR[92] R[102]% CNT100;
   1:  PR[91,1] = PR[90,1] + 36.477;
   1:  PR[91,2] = PR[90,2] + 36.392;
   1:  PR[92] = PR[91];
   1:  PR[92,3] = PR[92,3] + R[101];
   1:J PR[92] R[102]% CNT100;
   1:L PR[91] 100mm/sec FINE RampTo R[100]  Weld Start[1,5.0];
   1:  GO[2]=R[113];
   1:  PR[91,1] = PR[90,1] + 3.677;
   1:L PR[91] R[100]mm/sec CNT100;
   1:  PR[91,2] = PR[90,2] + 3.592;
   1:L PR[91] R[100]mm/sec CNT100;
   1:  PR[91,1] = PR[90,1] + 36.477;
   1:L PR[91] R[100]mm/sec CNT100;
   1:  PR[91,2] = PR[90,2] + 36.392;
   1:L PR[91] R[100]mm/sec CNT100  Weld End[1,5.0,0.2s];
   1:  WAIT R[104];
   1:  PR[92] = PR[91];
   1:  PR[92,3] = PR[92,3] + R[101];
   1:J PR[92] R[102]% CNT100;
   1:  PR[91,1] = PR[90,1] + 25.483;
   1:  PR[91,2] = PR[90,2] + 23.113;
   1:  PR[92] = PR[91];
   1:  PR[92,3] = PR[92,3] + R[101];
   1:J PR[92] R[102]% CNT100;
   1:L PR[91] 100mm/sec FINE RampTo R[100]  Weld Start[1,5.0];
   1:  GO[2]=R[113];
   1:  PR[91,1] = PR[90,1] + 26.320;
   1:  PR[91,2] = PR[90,2] + 19.992;
   1:L PR[91] R[100]mm/sec CNT100;
   1:  PR[91,1] = PR[90,1] + 25.483;
   1:  PR[91,2] = PR[90,2] + 16.870;
   1:L PR[91] R[100]mm/sec CNT100;
   1:  PR[91,1] = PR[90,1] + 23.198;
   1:  PR[91,2] = PR[90,2] + 14.586;
   1:L PR[91] R[100]mm/sec CNT100;
   1:  PR[91,1] = PR[90,1] + 20.077;
   1:  PR[91,2] = PR[90,2] + 13.750;
   1:L PR[91] R[100]mm/sec CNT100;
   1:  PR[91,1] = PR[90,1] + 16.957;
   1:  PR[91,2] = PR[90,2] + 14.586;
   1:L PR[91] R[100]mm/sec CNT100;
   1:  PR[91,1] = PR[90,1] + 14.672;
   1:  PR[91,2] = PR[90,2] + 16.870;
   1:L PR[91] R[100]mm/sec CNT100;
   1:  PR[91,1] = PR[90,1] + 13.835;
   1:  PR[91,2] = PR[90,2] + 19.992;
   1:L PR[91] R[100]mm/sec CNT100;
   1:  PR[91,1] = PR[90,1] + 14.672;
   1:  PR[91,2] = PR[90,2] + 23.113;
   1:L PR[91] R[100]mm/sec CNT100;
   1:  PR[91,1] = PR[90,1] + 16.957;
   1:  PR[91,2] = PR[90,2] + 25.398;
   1:L PR[91] R[100]mm/sec CNT100;
   1:  PR[91,1] = PR[90,1] + 20.077;
   1:  PR[91,2] = PR[90,2] + 26.234;
   1:L PR[91] R[100]mm/sec CNT100;
   1:  PR[91,1] = PR[90,1] + 23.198;
   1:  PR[91,2] = PR[90,2] + 25.398;
   1:L PR[91] R[100]mm/sec CNT100;
   1:  PR[91,1] = PR[90,1] + 25.483;
   1:  PR[91,2] = PR[90,2] + 23.113;
   1:L PR[91] R[100]mm/sec CNT100  Weld End[1,5.0,0.2s];
   1:  WAIT R[104];
   1:  PR[92] = PR[91];
   1:  PR[92,3] = PR[92,3] + R[101];
   1:J PR[92] R[102]% CNT100;
   1:  PR[91,1] = PR[90,1] + 27.635;
   1:  PR[91,2] = PR[90,2] + 24.356;
   1:  PR[92] = PR[91];
   1:  PR[92,3] = PR[92,3] + R[101];
   1:J PR[92] R[102]% CNT100;
   1:L PR[91] 100mm/sec FINE RampTo R[100]  Weld Start[1,5.0];
   1:  GO[2]=R[113];
   1:  PR[91,1] = PR[90,1] + 28.805;
   1:  PR[91,2] = PR[90,2] + 19.992;
   1:L PR[91] R[100]mm/sec CNT100;
   1:  PR[91,1] = PR[90,1] + 27.635;
   1:  PR[91,2] = PR[90,2] + 15.627;
   1:L PR[91] R[100]mm/sec CNT100;
   1:  PR[91,1] = PR[90,1] + 24.440;
   1:  PR[91,2] = PR[90,2] + 12.434;
   1:L PR[91] R[100]mm/sec CNT100;
   1:  PR[91,1] = PR[90,1] + 20.077;
   1:  PR[91,2] = PR[90,2] + 11.265;
   1:L PR[91] R[100]mm/sec CNT100;
   1:  PR[91,1] = PR[90,1] + 15.715;
   1:  PR[91,2] = PR[90,2] + 12.434;
   1:L PR[91] R[100]mm/sec CNT100;
   1:  PR[91,1] = PR[90,1] + 12.520;
   1:  PR[91,2] = PR[90,2] + 15.627;
   1:L PR[91] R[100]mm/sec CNT100;
   1:  PR[91,1] = PR[90,1] + 11.350;
   1:  PR[91,2] = PR[90,2] + 19.992;
   1:L PR[91] R[100]mm/sec CNT100;
   1:  PR[91,1] = PR[90,1] + 12.520;
   1:  PR[91,2] = PR[90,2] + 24.356;
   1:L PR[91] R[100]mm/sec CNT100;
   1:  PR[91,1] = PR[90,1] + 15.715;
   1:  PR[91,2] = PR[90,2] + 27.550;
   1:L PR[91] R[100]mm/sec CNT100;
   1:  PR[91,1] = PR[90,1] + 20.077;
   1:  PR[91,2] = PR[90,2] + 28.719;
   1:L PR[91] R[100]mm/sec CNT100;
   1:  PR[91,1] = PR[90,1] + 24.440;
   1:  PR[91,2] = PR[90,2] + 27.550;
   1:L PR[91] R[100]mm/sec CNT100;
   1:  PR[91,1] = PR[90,1] + 27.635;
   1:  PR[91,2] = PR[90,2] + 24.356;
   1:L PR[91] R[100]mm/sec CNT100  Weld End[1,5.0,0.2s];
   1:  WAIT R[104];
   1:  PR[92] = PR[91];
   1:  PR[92,3] = PR[92,3] + R[101];
   1:J PR[92] R[102]% CNT100;
   1:  PR[91,1] = PR[90,1] + 29.744;
   1:  PR[91,2] = PR[90,2] + 16.082;
   1:  PR[92] = PR[91];
   1:  PR[92,3] = PR[92,3] + R[101];
   1:J PR[92] R[102]% CNT100;
   1:L PR[91] 100mm/sec FINE RampTo R[100]  Weld Start[1,5.0];
   1:  GO[2]=R[113];
   1:  PR[91,1] = PR[90,1] + 34.557;
   1:  PR[91,2] = PR[90,2] + 20.895;
   1:L PR[91] R[100]mm/sec CNT100;
   1:  PR[91,2] = PR[90,2] + 24.289;
   1:L PR[91] R[100]mm/sec CNT100;
   1:  PR[91,1] = PR[90,1] + 30.680;
   1:  PR[91,2] = PR[90,2] + 20.412;
   1:L PR[91] R[100]mm/sec CNT100;
   1:  PR[91,1] = PR[90,1] + 29.962;
   1:  PR[91,2] = PR[90,2] + 23.088;
   1:L PR[91] R[100]mm/sec CNT100;
   1:  PR[91,1] = PR[90,1] + 34.557;
   1:  PR[91,2] = PR[90,2] + 27.683;
   1:L PR[91] R[100]mm/sec CNT100;
   1:  PR[91,2] = PR[90,2] + 31.078;
   1:L PR[91] R[100]mm/sec CNT100;
   1:  PR[91,1] = PR[90,1] + 29.093;
   1:  PR[91,2] = PR[90,2] + 25.613;
   1:L PR[91] R[100]mm/sec CNT100;
   1:  PR[91,1] = PR[90,1] + 27.396;
   1:  PR[91,2] = PR[90,2] + 27.310;
   1:L PR[91] R[100]mm/sec CNT100;
   1:  PR[91,1] = PR[90,1] + 34.557;
   1:  PR[91,2] = PR[90,2] + 34.472;
   1:L PR[91] R[100]mm/sec CNT100;
   1:  PR[91,1] = PR[90,1] + 31.163;
   1:L PR[91] R[100]mm/sec CNT100;
   1:  PR[91,1] = PR[90,1] + 25.698;
   1:  PR[91,2] = PR[90,2] + 29.007;
   1:L PR[91] R[100]mm/sec CNT100;
   1:  PR[91,1] = PR[90,1] + 25.434;
   1:  PR[91,2] = PR[90,2] + 29.271;
   1:L PR[91] R[100]mm/sec CNT100;
   1:  PR[91,1] = PR[90,1] + 23.174;
   1:  PR[91,2] = PR[90,2] + 29.877;
   1:L PR[91] R[100]mm/sec CNT100;
   1:  PR[91,1] = PR[90,1] + 27.769;
   1:  PR[91,2] = PR[90,2] + 34.472;
   1:L PR[91] R[100]mm/sec CNT100;
   1:  PR[91,1] = PR[90,1] + 24.375;
   1:L PR[91] R[100]mm/sec CNT100;
   1:  PR[91,1] = PR[90,1] + 20.497;
   1:  PR[91,2] = PR[90,2] + 30.594;
   1:L PR[91] R[100]mm/sec CNT100  Weld End[1,5.0,0.2s];
   1:  WAIT R[104];
   1:  PR[92] = PR[91];
   1:  PR[92,3] = PR[92,3] + R[101];
   1:J PR[92] R[102]% CNT100;
   1:  PR[91,1] = PR[90,1] + 7.405;
   1:  PR[91,2] = PR[90,2] + 34.472;
   1:  PR[92] = PR[91];
   1:  PR[92,3] = PR[92,3] + R[101];
   1:J PR[92] R[102]% CNT100;
   1:L PR[91] 100mm/sec FINE RampTo R[100]  Weld Start[1,5.0];
   1:  GO[2]=R[113];
   1:  PR[91,1] = PR[90,1] + 5.597;
   1:  PR[91,2] = PR[90,2] + 32.665;
   1:L PR[91] R[100]mm/sec CNT100;
   1:  PR[91,2] = PR[90,2] + 29.270;
   1:L PR[91] R[100]mm/sec CNT100;
   1:  PR[91,1] = PR[90,1] + 10.799;
   1:  PR[91,2] = PR[90,2] + 34.472;
   1:L PR[91] R[100]mm/sec CNT100;
   1:  PR[91,1] = PR[90,1] + 14.193;
   1:L PR[91] R[100]mm/sec CNT100;
   1:  PR[91,1] = PR[90,1] + 5.597;
   1:  PR[91,2] = PR[90,2] + 25.876;
   1:L PR[91] R[100]mm/sec CNT100;
   1:  PR[91,2] = PR[90,2] + 22.482;
   1:L PR[91] R[100]mm/sec CNT100;
   1:  PR[91,1] = PR[90,1] + 17.587;
   1:  PR[91,2] = PR[90,2] + 34.472;
   1:L PR[91] R[100]mm/sec CNT100;
   1:  PR[91,1] = PR[90,1] + 20.981;
   1:L PR[91] R[100]mm/sec CNT100;
   1:  PR[91,1] = PR[90,1] + 16.168;
   1:  PR[91,2] = PR[90,2] + 29.659;
   1:L PR[91] R[100]mm/sec CNT100;
   1:  PR[91,1] = PR[90,1] + 14.721;
   1:  PR[91,2] = PR[90,2] + 29.271;
   1:L PR[91] R[100]mm/sec CNT100;
   1:  PR[91,1] = PR[90,1] + 10.799;
   1:  PR[91,2] = PR[90,2] + 25.350;
   1:L PR[91] R[100]mm/sec CNT100;
   1:  PR[91,1] = PR[90,1] + 10.410;
   1:  PR[91,2] = PR[90,2] + 23.901;
   1:L PR[91] R[100]mm/sec CNT100;
   1:  PR[91,1] = PR[90,1] + 5.597;
   1:  PR[91,2] = PR[90,2] + 19.088;
   1:L PR[91] R[100]mm/sec CNT100;
   1:  PR[91,2] = PR[90,2] + 15.694;
   1:L PR[91] R[100]mm/sec CNT100;
   1:  PR[91,1] = PR[90,1] + 9.475;
   1:  PR[91,2] = PR[90,2] + 19.572;
   1:L PR[91] R[100]mm/sec CNT100;
   1:  PR[91,1] = PR[90,1] + 10.193;
   1:  PR[91,2] = PR[90,2] + 16.895;
   1:L PR[91] R[100]mm/sec CNT100;
   1:  PR[91,1] = PR[90,1] + 5.597;
   1:  PR[91,2] = PR[90,2] + 12.300;
   1:L PR[91] R[100]mm/sec CNT100;
   1:  PR[91,2] = PR[90,2] + 8.906;
   1:L PR[91] R[100]mm/sec CNT100;
   1:  PR[91,1] = PR[90,1] + 11.062;
   1:  PR[91,2] = PR[90,2] + 14.370;
   1:L PR[91] R[100]mm/sec CNT100;
   1:  PR[91,1] = PR[90,1] + 12.759;
   1:  PR[91,2] = PR[90,2] + 12.673;
   1:L PR[91] R[100]mm/sec CNT100;
   1:  PR[91,1] = PR[90,1] + 5.597;
   1:  PR[91,2] = PR[90,2] + 5.512;
   1:L PR[91] R[100]mm/sec CNT100;
   1:  PR[91,1] = PR[90,1] + 8.992;
   1:L PR[91] R[100]mm/sec CNT100;
   1:  PR[91,1] = PR[90,1] + 14.456;
   1:  PR[91,2] = PR[90,2] + 10.977;
   1:L PR[91] R[100]mm/sec CNT100;
   1:  PR[91,1] = PR[90,1] + 14.721;
   1:  PR[91,2] = PR[90,2] + 10.712;
   1:L PR[91] R[100]mm/sec CNT100;
   1:  PR[91,1] = PR[90,1] + 16.981;
   1:  PR[91,2] = PR[90,2] + 10.107;
   1:L PR[91] R[100]mm/sec CNT100;
   1:  PR[91,1] = PR[90,1] + 12.386;
   1:  PR[91,2] = PR[90,2] + 5.512;
   1:L PR[91] R[100]mm/sec CNT100;
   1:  PR[91,1] = PR[90,1] + 15.780;
   1:L PR[91] R[100]mm/sec CNT100;
   1:  PR[91,1] = PR[90,1] + 19.658;
   1:  PR[91,2] = PR[90,2] + 9.390;
   1:L PR[91] R[100]mm/sec CNT100;
   1:  PR[91,1] = PR[90,1] + 20.077;
   1:  PR[91,2] = PR[90,2] + 9.277;
   1:L PR[91] R[100]mm/sec CNT100;
   1:  PR[91,1] = PR[90,1] + 23.987;
   1:  PR[91,2] = PR[90,2] + 10.324;
   1:L PR[91] R[100]mm/sec CNT100;
   1:  PR[91,1] = PR[90,1] + 19.174;
   1:  PR[91,2] = PR[90,2] + 5.512;
   1:L PR[91] R[100]mm/sec CNT100;
   1:  PR[91,1] = PR[90,1] + 22.568;
   1:L PR[91] R[100]mm/sec CNT100;
   1:  PR[91,1] = PR[90,1] + 34.557;
   1:  PR[91,2] = PR[90,2] + 17.501;
   1:L PR[91] R[100]mm/sec CNT100;
   1:  PR[91,2] = PR[90,2] + 14.107;
   1:L PR[91] R[100]mm/sec CNT100;
   1:  PR[91,1] = PR[90,1] + 25.962;
   1:  PR[91,2] = PR[90,2] + 5.512;
   1:L PR[91] R[100]mm/sec CNT100;
   1:  PR[91,1] = PR[90,1] + 29.356;
   1:L PR[91] R[100]mm/sec CNT100;
   1:  PR[91,1] = PR[90,1] + 34.557;
   1:  PR[91,2] = PR[90,2] + 10.713;
   1:L PR[91] R[100]mm/sec CNT100;
   1:  PR[91,2] = PR[90,2] + 7.319;
   1:L PR[91] R[100]mm/sec CNT100;
   1:  PR[91,1] = PR[90,1] + 32.750;
   1:  PR[91,2] = PR[90,2] + 5.512;
   1:L PR[91] R[100]mm/sec CNT100  Weld End[1,5.0,0.2s];
   1:  PR[92] = PR[91];
   1:  PR[92,3] = PR[92,3] + 100;
   1:J PR[92] R[102]% CNT100;
   1:  WAIT   10.00(sec);
   1:  CALL HOME_ALL;
/POS
/END
